FUNCTION_BLOCK FB_HumiditySensor
VAR_INPUT
END_VAR
VAR_OUTPUT
END_VAR
VAR
	rHumidity : REAL;
	iRange : INT := 32767;
	iVmax : INT := 10;
	rZeroOffset : REAL := 0.95800;
	rSlope : REAL := 0.03068;
END_VAR

rHumidity := ((INT_TO_REAL(MyGVL.iInput1)/iRange)*iVmax - rZeroOffset)/rSlope;

PROPERTY getHumidity : REAL
GET
getHumidity := rHumidity;
END_GET
END_PROPERTY

END_FUNCTION_BLOCK

(* stored: Version 1.1.0.1, ProductVersion 3.1.4024.11
   POU FB_HumiditySensor: Id {900ae7ef-ff62-41aa-a512-a88f4015ca2e}, SpecialFunc None
   Property getHumidity: Id {15cf90e6-56c2-465b-8947-e07dd6a62a25}
   Get Get: Id {737b34dd-306f-4e55-a8c4-1d63e8717ea1} *)
